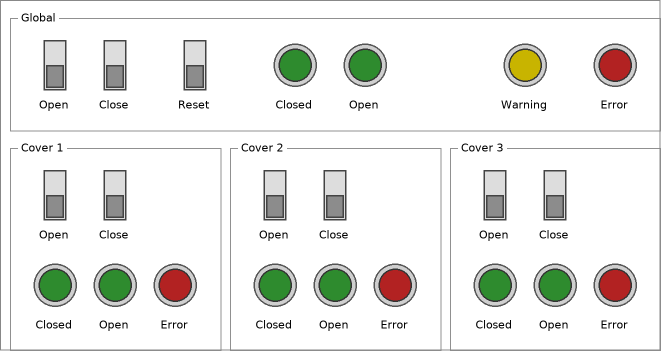
VISUALIZATION Cover  // 661x351
    GroupBox (10,10 651x121), "Global"
        DipSwitch (20,30 50x50), variable: MAIN.CoverControl.bOpen, behaviour: TOGGLE, style: Switch-DipSwitch-Gray
        DipSwitch (80,30 50x50), variable: MAIN.CoverControl.bClose, behaviour: TOGGLE, style: Switch-DipSwitch-Gray
        Lamp1 (260,30 50x50), variable: MAIN.CoverControl.bAllClosed, style: Lamp-Lamp1-Green
        Lamp1 (330,30 50x50), variable: MAIN.CoverControl.bAllOpen, style: Lamp-Lamp1-Green
        Label (10,80 68x30), "Open"
        Label (70,80 68x30), "Close"
        Label (250,80 68x30), "Closed"
        Label (320,80 68x30), "Open"
        DipSwitch (160,30 50x50), variable: MAIN.CoverControl.bReset, behaviour: TOGGLE, style: Switch-DipSwitch-Gray
        Lamp1 (490,30 50x50), variable: MAIN.CoverControl.bWarning, style: Lamp-Lamp1-Yellow
        Lamp1 (580,30 50x50), variable: MAIN.CoverControl.bError, style: Lamp-Lamp1-Red
        Label (570,80 68x30), "Error"
        Label (480,80 68x30), "Warning"
    GroupBox (10,140 211x211), "Cover 1"
        Label (130,170 68x30), "Error"
        Lamp1 (20,120 50x50), variable: MAIN.CoverControl.abCoverClosed[1], style: Lamp-Lamp1-Green
        Lamp1 (80,120 50x50), variable: MAIN.CoverControl.abCoverOpen[1], style: Lamp-Lamp1-Green
        Label (10,170 68x30), "Closed"
        Label (70,170 68x30), "Open"
        DipSwitch (20,30 50x50), variable: MAIN.CoverControl.OabOpenCover[1], behaviour: TOGGLE, style: Switch-DipSwitch-Gray
        DipSwitch (80,30 50x50), variable: MAIN.CoverControl.OabCloseCover[1], behaviour: TOGGLE, style: Switch-DipSwitch-Gray
        Label (10,80 68x30), "Open"
        Label (70,80 68x30), "Close"
        Lamp1 (140,120 50x50), variable: MAIN.CoverControl.abCoverError[1], style: Lamp-Lamp1-Red
    Label (160,90 68x30), "Reset"
    GroupBox (230,140 211x211), "Cover 2"
        Label (130,170 68x30), "Error"
        Lamp1 (20,120 50x50), variable: MAIN.CoverControl.abCoverClosed[2], style: Lamp-Lamp1-Green
        Lamp1 (80,120 50x50), variable: MAIN.CoverControl.abCoverOpen[2], style: Lamp-Lamp1-Green
        Label (10,170 68x30), "Closed"
        Label (70,170 68x30), "Open"
        DipSwitch (20,30 50x50), variable: MAIN.CoverControl.OabOpenCover[2], behaviour: TOGGLE, style: Switch-DipSwitch-Gray
        DipSwitch (80,30 50x50), variable: MAIN.CoverControl.OabCloseCover[2], behaviour: TOGGLE, style: Switch-DipSwitch-Gray
        Label (10,80 68x30), "Open"
        Label (70,80 68x30), "Close"
        Lamp1 (140,120 50x50), variable: MAIN.CoverControl.abCoverError[2], style: Lamp-Lamp1-Red
    GroupBox (450,140 211x211), "Cover 3"
        Label (130,170 68x30), "Error"
        Lamp1 (20,120 50x50), variable: MAIN.CoverControl.abCoverClosed[3], style: Lamp-Lamp1-Green
        Lamp1 (80,120 50x50), variable: MAIN.CoverControl.abCoverOpen[3], style: Lamp-Lamp1-Green
        Label (10,170 68x30), "Closed"
        Label (70,170 68x30), "Open"
        DipSwitch (20,30 50x50), variable: MAIN.CoverControl.OabOpenCover[3], behaviour: TOGGLE, style: Switch-DipSwitch-Gray
        DipSwitch (80,30 50x50), variable: MAIN.CoverControl.OabCloseCover[3], behaviour: TOGGLE, style: Switch-DipSwitch-Gray
        Label (10,80 68x30), "Open"
        Label (70,80 68x30), "Close"
        Lamp1 (140,120 50x50), variable: MAIN.CoverControl.abCoverError[3], style: Lamp-Lamp1-Red
END_VISUALIZATION

(* stored: Version 1.1.0.1, ProductVersion 3.1.4024.15
   Visu Cover: Id {b255d8a6-76d1-4ce0-8ffb-0acc65fd87df} *)
